FUNCTION_BLOCK MECH2_SVR (* Bidirectional Mechanism Server for a Remote MECH2_PRXY *)
  (* Standard: 61499-1 *)
  (* Version 0.0, 2004-09-26, JHC, Rockwell Automation *)
  (* Compiler header: package fb.rt.mva; import fb.rt.net.*; *)
  (* Compiler Java Sun JDK 1.4.2 *)
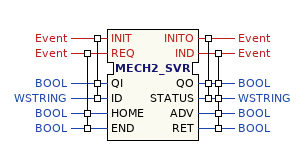
  EVENT_INPUT
    INIT WITH QI, ID; (* Initialize Client/Server Connection *)
    REQ WITH HOME, END; (* Send Sensor Data *)
  END_EVENT
  EVENT_OUTPUT
    INITO WITH QO, STATUS; (* INIT Acknowledgment *)
    IND WITH ADV, RET, QO, STATUS; (* Actuator Change Indication *)
  END_EVENT
  VAR_INPUT
    QI : BOOL; (* Event Input Qualifier *)
    ID : WSTRING; (* Connection Identifier *)
    HOME : BOOL; (* HOME Position Sensor *)
    END : BOOL; (* END Position Sensor *)
  END_VAR
  VAR_OUTPUT
    QO : BOOL; (* Event Output Qualifier *)
    STATUS : WSTRING; (* Service Status *)
    ADV : BOOL; (* ADVANCE *)
    RET : BOOL; (* RETRACT *)
  END_VAR
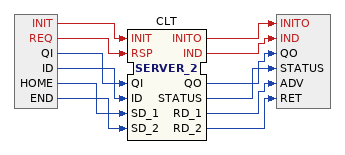
  FBS
    CLT : SERVER_2;
  END_FBS
  EVENT_CONNECTIONS
    INIT TO CLT.INIT;
    CLT.INITO TO INITO;
    CLT.IND TO IND;
    REQ TO CLT.RSP;
  END_CONNECTIONS
  DATA_CONNECTIONS
    QI TO CLT.QI;
    CLT.QO TO QO;
    ID TO CLT.ID;
    CLT.STATUS TO STATUS;
    HOME TO CLT.SD_1;
    END TO CLT.SD_2;
    CLT.RD_1 TO ADV;
    CLT.RD_2 TO RET;
  END_CONNECTIONS
END_FUNCTION_BLOCK
